// TIA Portal V16 export
// export: Created 2021-05-25T16:14:35.0542513Z, ExportSetting WithDefaults, DisplayName Totally Integrated Automation Portal, DisplayVersion V16, DisplayName TIA Portal Version Control Interface, DisplayVersion V16, DisplayName TIA Portal Openness, DisplayVersion V16, DisplayName STEP 7 Professional, DisplayVersion V16, DisplayName STEP 7 Safety, DisplayVersion V16, DisplayName WinCC Unified SCADA Engineering System, DisplayVersion V16
DATA_BLOCK "ph_LegsShifter_2_DB"   // DB311
VERSION : 0.1
// stored: AutoNumber false, DBAccessibleFromOPCUA true, InstanceOfName ph_LegsShifter_2, InstanceOfType FB
"ph_LegsShifter_2"
   // VAR_IN_OUT
   //    Y17_RotCilipozDesno : "udtDigitalValve";
   //    Y18_RotCilipozLevo : "udtDigitalValve";
   //    Y6_DrcaLocev_Des : "udtDigitalValve";
   //    Y7_DrcaLocev_Lev : "udtDigitalValve";
   // END_VAR
   // VAR RETAIN
   //    CurrentStep { ExternalAccessible := 'False'; ExternalVisible := 'False'; ExternalWritable := 'False'} : Int := 0;
   //    PhaseStatus { ExternalAccessible := 'False'; ExternalVisible := 'False'; ExternalWritable := 'False'} : Int := 0;
   //    Mode { ExternalAccessible := 'False'; ExternalVisible := 'False'; ExternalWritable := 'False'} : SInt := 2;
   //    AlarmPresent { ExternalAccessible := 'False'; ExternalVisible := 'False'; ExternalWritable := 'False'} : Bool := FALSE;
   //    InitPosition { ExternalAccessible := 'False'; ExternalVisible := 'False'; ExternalWritable := 'False'} : Bool := TRUE;
   // END_VAR
   // VAR
   //    StartCmd { ExternalAccessible := 'False'; ExternalVisible := 'False'; ExternalWritable := 'False'} : Bool := FALSE;
   //    AlarmPresentOLD { ExternalAccessible := 'False'; ExternalVisible := 'False'; ExternalWritable := 'False'} : Bool := FALSE;
   //    InitPositionOLD { ExternalAccessible := 'False'; ExternalVisible := 'False'; ExternalWritable := 'False'} : Bool := TRUE;
   //    IEC_TimerOnDly_1 { ExternalAccessible := 'False'; ExternalVisible := 'False'; ExternalWritable := 'False'} : TONR_TIME;
   //    IEC_TimerOnDly_2 { ExternalAccessible := 'False'; ExternalVisible := 'False'; ExternalWritable := 'False'} : TONR_TIME;
   //    IEC_TimerOnDly_3 { ExternalAccessible := 'False'; ExternalVisible := 'False'; ExternalWritable := 'False'} : TONR_TIME;
   //    IEC_TimerOnDly_4 { ExternalAccessible := 'False'; ExternalVisible := 'False'; ExternalWritable := 'False'} : TONR_TIME;
   //    IEC_TimerOnDly_5 { ExternalAccessible := 'False'; ExternalVisible := 'False'; ExternalWritable := 'False'} : TONR_TIME;
   //    IEC_TimerOnDly_6 { ExternalAccessible := 'False'; ExternalVisible := 'False'; ExternalWritable := 'False'} : TONR_TIME;
   //    IEC_TimerOnDly_7 { ExternalAccessible := 'False'; ExternalVisible := 'False'; ExternalWritable := 'False'} : TONR_TIME;
   //    IEC_TimerOnDly_8 { ExternalAccessible := 'False'; ExternalVisible := 'False'; ExternalWritable := 'False'} : TONR_TIME;
   //    IEC_TimerOnDly_9 { ExternalAccessible := 'False'; ExternalVisible := 'False'; ExternalWritable := 'False'} : TONR_TIME;
   //    IEC_TimerOnDly_10 { ExternalAccessible := 'False'; ExternalVisible := 'False'; ExternalWritable := 'False'} : TONR_TIME;
   //    IEC_TimerOnDly_ET_1 { ExternalAccessible := 'False'; ExternalVisible := 'False'; ExternalWritable := 'False'} : Time := T#0MS;
   //    IEC_TimerOnDly_ET_2 { ExternalAccessible := 'False'; ExternalVisible := 'False'; ExternalWritable := 'False'} : Time := T#0MS;
   //    IEC_TimerOnDly_ET_3 { ExternalAccessible := 'False'; ExternalVisible := 'False'; ExternalWritable := 'False'} : Time := T#0MS;
   //    IEC_TimerOnDly_ET_4 { ExternalAccessible := 'False'; ExternalVisible := 'False'; ExternalWritable := 'False'} : Time := T#0MS;
   //    IEC_TimerOnDly_ET_5 { ExternalAccessible := 'False'; ExternalVisible := 'False'; ExternalWritable := 'False'} : Time := T#0MS;
   //    IEC_TimerOnDly_ET_6 { ExternalAccessible := 'False'; ExternalVisible := 'False'; ExternalWritable := 'False'} : Time := T#0MS;
   //    IEC_TimerOnDly_ET_7 { ExternalAccessible := 'False'; ExternalVisible := 'False'; ExternalWritable := 'False'} : Time := T#0MS;
   //    IEC_TimerOnDly_ET_8 { ExternalAccessible := 'False'; ExternalVisible := 'False'; ExternalWritable := 'False'} : Time := T#0MS;
   //    IEC_TimerOnDly_ET_9 { ExternalAccessible := 'False'; ExternalVisible := 'False'; ExternalWritable := 'False'} : Time := T#0MS;
   //    IEC_TimerOnDly_ET_10 { ExternalAccessible := 'False'; ExternalVisible := 'False'; ExternalWritable := 'False'} : Time := T#0MS;
   //    IEC_TimerOnDly_DN_1 { ExternalAccessible := 'False'; ExternalVisible := 'False'; ExternalWritable := 'False'} : Bool := FALSE;
   //    IEC_TimerOnDly_DN_2 { ExternalAccessible := 'False'; ExternalVisible := 'False'; ExternalWritable := 'False'} : Bool := FALSE;
   //    IEC_TimerOnDly_DN_3 { ExternalAccessible := 'False'; ExternalVisible := 'False'; ExternalWritable := 'False'} : Bool := FALSE;
   //    IEC_TimerOnDly_DN_4 { ExternalAccessible := 'False'; ExternalVisible := 'False'; ExternalWritable := 'False'} : Bool := FALSE;
   //    IEC_TimerOnDly_DN_5 { ExternalAccessible := 'False'; ExternalVisible := 'False'; ExternalWritable := 'False'} : Bool := FALSE;
   //    IEC_TimerOnDly_DN_6 { ExternalAccessible := 'False'; ExternalVisible := 'False'; ExternalWritable := 'False'} : Bool := FALSE;
   //    IEC_TimerOnDly_DN_7 { ExternalAccessible := 'False'; ExternalVisible := 'False'; ExternalWritable := 'False'} : Bool := FALSE;
   //    IEC_TimerOnDly_DN_8 { ExternalAccessible := 'False'; ExternalVisible := 'False'; ExternalWritable := 'False'} : Bool := FALSE;
   //    IEC_TimerOnDly_DN_9 { ExternalAccessible := 'False'; ExternalVisible := 'False'; ExternalWritable := 'False'} : Bool := FALSE;
   //    IEC_TimerOnDly_DN_10 { ExternalAccessible := 'False'; ExternalVisible := 'False'; ExternalWritable := 'False'} : Bool := FALSE;
   //    FillingLineSelector { ExternalAccessible := 'False'; ExternalVisible := 'False'; ExternalWritable := 'False'} : USInt := 1;
   //    InletLineStep { ExternalAccessible := 'False'; ExternalVisible := 'False'; ExternalWritable := 'False'} : SInt := 2;
   //    LeftOutletLineStep { ExternalAccessible := 'False'; ExternalVisible := 'False'; ExternalWritable := 'False'} : SInt := 0;
   //    RightOutletLineStep { ExternalAccessible := 'False'; ExternalVisible := 'False'; ExternalWritable := 'False'} : SInt := 0;
   // END_VAR
   // VAR RETAIN
   //    TimeToLoadInletLine { S7_SetPoint := 'True'} : Int := 15;
   //    TimeToReleaseInletLine { S7_SetPoint := 'True'} : Int := 15;
   //    TimeToReleaseOutletLine { S7_SetPoint := 'True'} : Int := 10;
   // END_VAR
   // VAR
   //    LeftLegIndex { ExternalAccessible := 'False'; ExternalVisible := 'False'; ExternalWritable := 'False'} : SInt := 2;
   //    RightLegIndex { ExternalAccessible := 'False'; ExternalVisible := 'False'; ExternalWritable := 'False'} : SInt := 2;
   //    LeftFirstLegIndex { ExternalAccessible := 'False'; ExternalVisible := 'False'; ExternalWritable := 'False'} : SInt := 2;
   //    RightFirstLegIndex { ExternalAccessible := 'False'; ExternalVisible := 'False'; ExternalWritable := 'False'} : SInt := 2;
   //    DRCA_DESNO_LATCH { ExternalAccessible := 'False'; ExternalVisible := 'False'; ExternalWritable := 'False'} : Bool := FALSE;
   //    DRCA_LEVO_LATCH { ExternalAccessible := 'False'; ExternalVisible := 'False'; ExternalWritable := 'False'} : Bool := FALSE;
   // END_VAR
BEGIN
   IEC_TimerOnDly_1.PT := T#0MS;
   IEC_TimerOnDly_1.IN := FALSE;
   IEC_TimerOnDly_2.PT := T#0MS;
   IEC_TimerOnDly_2.IN := FALSE;
   IEC_TimerOnDly_3.PT := T#0MS;
   IEC_TimerOnDly_3.IN := FALSE;
   IEC_TimerOnDly_4.PT := T#0MS;
   IEC_TimerOnDly_4.IN := FALSE;
   IEC_TimerOnDly_5.PT := T#0MS;
   IEC_TimerOnDly_5.IN := FALSE;
   IEC_TimerOnDly_6.PT := T#0MS;
   IEC_TimerOnDly_6.IN := FALSE;
   IEC_TimerOnDly_7.PT := T#0MS;
   IEC_TimerOnDly_7.IN := FALSE;
   IEC_TimerOnDly_8.PT := T#0MS;
   IEC_TimerOnDly_8.IN := FALSE;
   IEC_TimerOnDly_9.PT := T#0MS;
   IEC_TimerOnDly_9.IN := FALSE;
   IEC_TimerOnDly_10.PT := T#0MS;
   IEC_TimerOnDly_10.IN := FALSE;
END_DATA_BLOCK
